INTERFACE I_ServerResponse

METHOD PUBLIC Accepted
VAR_INPUT
END_VAR
END_METHOD

METHOD PUBLIC Busy
VAR_INPUT
END_VAR
END_METHOD

METHOD PUBLIC Error
VAR_INPUT
	Message : T_MAXSTRING;
END_VAR
END_METHOD

PROPERTY PUBLIC Header : I_Header
GET
END_GET
END_PROPERTY

PROPERTY PUBLIC HeadersSent : BOOL
GET
END_GET
END_PROPERTY

METHOD PUBLIC Pending
VAR_INPUT
	ResponseId : REFERENCE TO T_MAXSTRING;
	RetryDelayInMs : UDINT;
END_VAR
END_METHOD

METHOD PUBLIC Success
VAR_INPUT
END_VAR
END_METHOD

METHOD PUBLIC SuccessWithPayload
VAR_INPUT
	PayloadDataAddress : PVOID;
	PayloadDataSize : UDINT;
END_VAR
END_METHOD

END_INTERFACE

(* stored: Version 1.1.0.1, ProductVersion 3.1.4024.12
   Itf I_ServerResponse: Id {e7875b2f-2f6c-491d-bc7c-66dc808265d5}
   Method Accepted: Id {5da939c4-cc98-4864-8b65-87bfcd25a1cc}
   Method Busy: Id {375082fc-ee95-407c-aff4-a51f39c86f1f}
   Method Error: Id {1a106d6d-2b14-4d9c-a03e-2cffd9200ec6}
   Property Header: Id {e4fcf1e6-4e4e-4543-82d0-51f8c8a85113}
   Get Get: Id {67cd667d-6708-4212-ac18-80548d414748}
   Property HeadersSent: Id {49c401e6-f7fd-4286-a646-e1ea83bd5c11}
   Get Get: Id {d5bb7f3f-9691-4516-adcd-cf4093e1bb40}
   Method Pending: Id {bdb38a65-0216-448e-94dc-5962ebc5f820}
   Method Success: Id {dcba0e73-d1db-4767-a918-598bfb8da5cb}
   Method SuccessWithPayload: Id {8212960f-67a8-4f5b-b6a5-06afdb71fe7e} *)
